TYPE ST_SimulinkModel_forControl_Output :
STRUCT
	Disp_P: matrix_18_real_T;
END_STRUCT
END_TYPE

(* stored: Version 1.1.0.1, ProductVersion 3.1.4020.12
   DUT ST_SimulinkModel_forControl_Output: Id {948ee725-58fa-4f71-ab9d-aea6c0198018} *)
